INTERFACE I_EventDetailer

METHOD GetDetail : STRING(255)
VAR_INPUT
	TcAlarm : REFERENCE TO FB_TcAlarm;
END_VAR
END_METHOD

END_INTERFACE

(* stored: Version 1.1.0.1, ProductVersion 3.1.4024.13
   Itf I_EventDetailer: Id {6f69f0dc-e3bf-4582-9e64-540faae44557}
   Method GetDetail: Id {44338422-a1ab-455f-bb4e-b66cc24ed120} *)
